PROGRAM Axis05_Manual
VAR
	Always_ON	:	BOOL	:=TRUE	;//상시 ON 
	Always_OFF	:	BOOL	:=FALSE	;//상시 OFF
END_VAR

// NETWORK 1

END_PROGRAM

(* stored: Version 1.1.0.1, ProductVersion 3.1.4024.15
   POU Axis05_Manual: Id {9e769e66-efb3-499d-8b36-05e79ce2e9bc}, SpecialFunc None *)
